FUNCTION_BLOCK FB_AstroClock
VAR_INPUT
END_VAR
VAR_OUTPUT
        time_RTCEX      : DT;
        time_RTCEX2     : TIMESTRUCT;
        nMilliseconds   : DWORD;
        nMicroseconds   : DWORD;
END_VAR
VAR
	        fbGetLocalTime  : NT_GetTime;
        bBusy           : BOOL;
        bError          : BOOL;
        nErrID          : UDINT;
        presetTime      : TIMESTRUCT;

        syncTimer       : TON;
        syncTrigger     : F_TRIG;
        bSynchronize    : BOOL;

        fbRTC           : RTC;
        bValid_RTC      : BOOL;
        time_RTC        : DT;

        fbRTC_EX        : RTC_EX;
        bValid_RTCEX    : BOOL;

        fbRTC_EX2       : RTC_EX2;
        bValid_RTCEX2   : BOOL;
END_VAR

(*
TYPE TIMESTRUCT
STRUCT
   wYear            : WORD;
   wMonth           : WORD;
   wDayOfWeek       : WORD;
   wDay             : WORD;
   wHour            : WORD;
   wMinute          : WORD;
   wSecond          : WORD;
   wMilliseconds    : WORD;
END_STRUCT
END_TYPE
*)

syncTimer(IN := NOT SyncTimer.Q, PT := T#5S);
fbGetLocalTime(START := syncTimer.Q,
	TMOUT := DEFAULT_ADS_TIMEOUT,
	Busy => bBusy,
	ERR => bError,
	ERRID => nErrID,
	TIMESTR => presetTime);

syncTrigger(CLK := bBusy AND NOT bError, Q => bSynchronize);

fbRTC(EN := bSynchronize,
	PDT := SYSTEMTIME_TO_DT(presetTime),
	Q => bValid_RTC,
	CDT => time_RTC);
	
fbRTC_EX(EN := bSynchronize,
	PDT := SYSTEMTIME_TO_DT(presetTime),
	PMSEK := presetTime.wMilliseconds,
	Q => bValid_RTCEX,
	CDT => time_RTCEX,
	CMSEK => nMilliseconds);

fbRTC_EX2(EN := bSynchronize,
	PDT := presetTime,
	PMICRO := 0,
	Q => bValid_RTCEX2,
	CDT => time_RTCEX2,
	CMICRO => nMicroseconds);

END_FUNCTION_BLOCK

(* stored: Version 1.1.0.1, ProductVersion 3.1.4024.4
   POU FB_AstroClock: Id {9eeab12b-19b9-408a-b96c-52351be0dfa7}, SpecialFunc None *)
